(*
SPDX-FileCopyrightText: © 2026 Oleksandr Tiutyk <trofimich@gmail.com>
SPDX-License-Identifier: MIT
License: https://opensource.org/license/mit
*)

{attribute 'qualified_only'}
{attribute 'strict'}
{attribute 'to_string'}
TYPE LOGICAL_OPERATOR :
(
	AND_ := 0,
	OR_ := 1
) BYTE;
END_TYPE

(* stored: Version 1.1.0.1
   DUT LOGICAL_OPERATOR: Id {858be361-e7f2-4b47-bbf7-3e230569860c} *)
